Staubli VAL3: new.pgx

public program new(string x_sItem, num x_nIndex)
begin
  // insert a new item
  //insert(saveAxis[x_nIndex])
  $dins(nSaveaxis,size(nSaveaxis))
  $dins(nSaveaxis1,size(nSaveaxis1))
  $dins(sSaveaxis,size(sSaveaxis))
  $dins(nVelocity,size(nVelocity))
  sSaveaxis[size(sSaveaxis)-1]=x_sItem
  nVelocity[size(nVelocity)-1]=8
  ? x_sItem
end
